FUNCTION_BLOCK Recipe_10010_transportreserve_1
VAR_INPUT
	execute	: BOOL;
	Order	: DUT_RECIPEORDER;
END_VAR
VAR_OUTPUT
	RecipeInfo	: DUT_RECIPEOFFER;
	RecipeDone	: BOOL;	
	InitDone	: BOOL;
END_VAR
VAR
	StepDone	: BOOL;
END_VAR

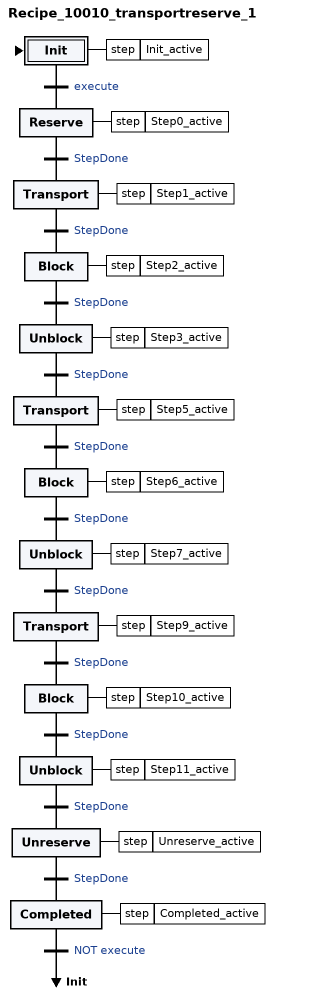
INITIAL_STEP Init:
    Init_active(N);  // step action
END_STEP
TRANSITION FROM Init TO Reserve
    := execute;
END_TRANSITION
STEP Reserve:
    Step0_active(N);  // step action
END_STEP
TRANSITION FROM Reserve TO Transport
    := StepDone;
END_TRANSITION
STEP Transport:
    Step1_active(N);  // step action
END_STEP
TRANSITION FROM Transport TO Block
    := StepDone;
END_TRANSITION
STEP Block:
    Step2_active(N);  // step action
END_STEP
TRANSITION FROM Block TO Unblock
    := StepDone;
END_TRANSITION
STEP Unblock:
    Step3_active(N);  // step action
END_STEP
TRANSITION FROM Unblock TO Transport
    := StepDone;
END_TRANSITION
STEP Transport:
    Step5_active(N);  // step action
END_STEP
TRANSITION FROM Transport TO Block
    := StepDone;
END_TRANSITION
STEP Block:
    Step6_active(N);  // step action
END_STEP
TRANSITION FROM Block TO Unblock
    := StepDone;
END_TRANSITION
STEP Unblock:
    Step7_active(N);  // step action
END_STEP
TRANSITION FROM Unblock TO Transport
    := StepDone;
END_TRANSITION
STEP Transport:
    Step9_active(N);  // step action
END_STEP
TRANSITION FROM Transport TO Block
    := StepDone;
END_TRANSITION
STEP Block:
    Step10_active(N);  // step action
END_STEP
TRANSITION FROM Block TO Unblock
    := StepDone;
END_TRANSITION
STEP Unblock:
    Step11_active(N);  // step action
END_STEP
TRANSITION FROM Unblock TO Unreserve
    := StepDone;
END_TRANSITION
STEP Unreserve:
    Unreserve_active(N);  // step action
END_STEP
TRANSITION FROM Unreserve TO Completed
    := StepDone;
END_TRANSITION
STEP Completed:
    Completed_active(N);  // step action
END_STEP
TRANSITION FROM Completed TO Init
    := NOT execute;
END_TRANSITION

ACTION Block_active:
StepDone := FALSE;

//Skill auswählen
ExecuteSkill.SkillID 		:= 1315;
ExecuteSkill.SkillName	 	:= 'Block';

//Parameter setzen

ExecuteSkill.Parameter[1].ID := 1;
ExecuteSkill.Parameter[1].Name := 'TaskID';
ExecuteSkill.Parameter[1].Value := 124;


(*
ExecuteSkill.Parameter[2].ID := ;
ExecuteSkill.Parameter[2].Name := '';
ExecuteSkill.Parameter[2].Value := ;
*)

(*
ExecuteSkill.Parameter[3].ID := ;
ExecuteSkill.Parameter[3].Name := '';
ExecuteSkill.Parameter[3].Value := ;
*)

(*
ExecuteSkill.Parameter[4].ID := ;
ExecuteSkill.Parameter[4].Name := '';
ExecuteSkill.Parameter[4].Value := ;
*)

(*
ExecuteSkill.Parameter[5].ID := ;
ExecuteSkill.Parameter[5].Name := '';
ExecuteSkill.Parameter[5].Value := ;
*)



ExecuteSkill();

StepDone := ExecuteSkill.Done;
END_ACTION

ACTION Unreserve_active:
StepDone := FALSE;

//Skill auswählen
ExecuteSkill.SkillID 		:= 1311;
ExecuteSkill.SkillName	 	:= 'Unreserve';

//Parameter setzen

ExecuteSkill.Parameter[1].ID := 1;
ExecuteSkill.Parameter[1].Name := 'TaskID';
ExecuteSkill.Parameter[1].Value := 131;


(*
ExecuteSkill.Parameter[2].ID := ;
ExecuteSkill.Parameter[2].Name := '';
ExecuteSkill.Parameter[2].Value := ;
*)

(*
ExecuteSkill.Parameter[3].ID := ;
ExecuteSkill.Parameter[3].Name := '';
ExecuteSkill.Parameter[3].Value := ;
*)

(*
ExecuteSkill.Parameter[4].ID := ;
ExecuteSkill.Parameter[4].Name := '';
ExecuteSkill.Parameter[4].Value := ;
*)

(*
ExecuteSkill.Parameter[5].ID := ;
ExecuteSkill.Parameter[5].Name := '';
ExecuteSkill.Parameter[5].Value := ;
*)



ExecuteSkill();

StepDone := ExecuteSkill.Done;
END_ACTION

ACTION Unblock_active:
StepDone := FALSE;

//Skill auswählen
ExecuteSkill.SkillID 		:= 1316;
ExecuteSkill.SkillName	 	:= 'Unblock';

//Parameter setzen

ExecuteSkill.Parameter[1].ID := 1;
ExecuteSkill.Parameter[1].Name := 'TaskID';
ExecuteSkill.Parameter[1].Value := 125;


(*
ExecuteSkill.Parameter[2].ID := ;
ExecuteSkill.Parameter[2].Name := '';
ExecuteSkill.Parameter[2].Value := ;
*)

(*
ExecuteSkill.Parameter[3].ID := ;
ExecuteSkill.Parameter[3].Name := '';
ExecuteSkill.Parameter[3].Value := ;
*)

(*
ExecuteSkill.Parameter[4].ID := ;
ExecuteSkill.Parameter[4].Name := '';
ExecuteSkill.Parameter[4].Value := ;
*)

(*
ExecuteSkill.Parameter[5].ID := ;
ExecuteSkill.Parameter[5].Name := '';
ExecuteSkill.Parameter[5].Value := ;
*)



ExecuteSkill();

StepDone := ExecuteSkill.Done;
END_ACTION

ACTION Transport1_active:
StepDone := FALSE;

//Skill auswählen
ExecuteSkill.SkillID 		:= 1320;
ExecuteSkill.SkillName	 	:= 'Name';

//Parameter setzen

ExecuteSkill.Parameter[1].ID := 3;
ExecuteSkill.Parameter[1].Name := 'Velocity';
ExecuteSkill.Parameter[1].Value := 2500;



ExecuteSkill.Parameter[2].ID := 4 ;
ExecuteSkill.Parameter[2].Name := 'Acceleration';
ExecuteSkill.Parameter[2].Value := 1000 ;



ExecuteSkill.Parameter[3].ID := 1;
ExecuteSkill.Parameter[3].Name := 'TargetPosition X';
ExecuteSkill.Parameter[3].Value := 3200 ;



ExecuteSkill.Parameter[4].ID := 2;
ExecuteSkill.Parameter[4].Name := 'TargetPosition Z';
ExecuteSkill.Parameter[4].Value := 65 ;


(*
ExecuteSkill.Parameter[5].ID := ;
ExecuteSkill.Parameter[5].Name := '';
ExecuteSkill.Parameter[5].Value := ;
*)



ExecuteSkill();

StepDone := ExecuteSkill.Done;
END_ACTION

ACTION Block1_active:
StepDone := FALSE;

//Skill auswählen
ExecuteSkill.SkillID 		:= 1315;
ExecuteSkill.SkillName	 	:= 'Block';

//Parameter setzen

ExecuteSkill.Parameter[1].ID := 1;
ExecuteSkill.Parameter[1].Name := 'TaskID';
ExecuteSkill.Parameter[1].Value := 127;


(*
ExecuteSkill.Parameter[2].ID := ;
ExecuteSkill.Parameter[2].Name := '';
ExecuteSkill.Parameter[2].Value := ;
*)

(*
ExecuteSkill.Parameter[3].ID := ;
ExecuteSkill.Parameter[3].Name := '';
ExecuteSkill.Parameter[3].Value := ;
*)

(*
ExecuteSkill.Parameter[4].ID := ;
ExecuteSkill.Parameter[4].Name := '';
ExecuteSkill.Parameter[4].Value := ;
*)

(*
ExecuteSkill.Parameter[5].ID := ;
ExecuteSkill.Parameter[5].Name := '';
ExecuteSkill.Parameter[5].Value := ;
*)



ExecuteSkill();

StepDone := ExecuteSkill.Done;
END_ACTION

ACTION Reserve_active:
StepDone := FALSE;
RecipeDone := FALSE;
//Skill auswählen
ExecuteSkill.SkillID 		:= 1310;
ExecuteSkill.SkillName	 	:= 'Reserve';

//Parameter setzen

ExecuteSkill.Parameter[1].ID := 1;
ExecuteSkill.Parameter[1].Name := 'TaskID';
ExecuteSkill.Parameter[1].Value := 123;


(*
ExecuteSkill.Parameter[2].ID := ;
ExecuteSkill.Parameter[2].Name := '';
ExecuteSkill.Parameter[2].Value := ;
*)

(*
ExecuteSkill.Parameter[3].ID := ;
ExecuteSkill.Parameter[3].Name := '';
ExecuteSkill.Parameter[3].Value := ;
*)

(*
ExecuteSkill.Parameter[4].ID := ;
ExecuteSkill.Parameter[4].Name := '';
ExecuteSkill.Parameter[4].Value := ;
*)

(*
ExecuteSkill.Parameter[5].ID := ;
ExecuteSkill.Parameter[5].Name := '';
ExecuteSkill.Parameter[5].Value := ;
*)



ExecuteSkill();

StepDone := ExecuteSkill.Done;
END_ACTION

ACTION Completed_active:
RecipeDone := TRUE;
StepDone := FALSE;
END_ACTION

ACTION Unblock1_active:
StepDone := FALSE;

//Skill auswählen
ExecuteSkill.SkillID 		:= 1316;
ExecuteSkill.SkillName	 	:= 'Unblock';

//Parameter setzen

ExecuteSkill.Parameter[1].ID := 1;
ExecuteSkill.Parameter[1].Name := 'TaskID';
ExecuteSkill.Parameter[1].Value := 128 ;


(*
ExecuteSkill.Parameter[2].ID := ;
ExecuteSkill.Parameter[2].Name := '';
ExecuteSkill.Parameter[2].Value := ;
*)

(*
ExecuteSkill.Parameter[3].ID := ;
ExecuteSkill.Parameter[3].Name := '';
ExecuteSkill.Parameter[3].Value := ;
*)

(*
ExecuteSkill.Parameter[4].ID := ;
ExecuteSkill.Parameter[4].Name := '';
ExecuteSkill.Parameter[4].Value := ;
*)

(*
ExecuteSkill.Parameter[5].ID := ;
ExecuteSkill.Parameter[5].Name := '';
ExecuteSkill.Parameter[5].Value := ;
*)



ExecuteSkill();

StepDone := ExecuteSkill.Done;
END_ACTION

ACTION Transport2_active:
StepDone := FALSE;

//Skill auswählen
ExecuteSkill.SkillID 		:= 1320;
ExecuteSkill.SkillName	 	:= 'Transport';

//Parameter setzen

ExecuteSkill.Parameter[1].ID := 3;
ExecuteSkill.Parameter[1].Name := 'Velocity';
ExecuteSkill.Parameter[1].Value := 2800;



ExecuteSkill.Parameter[2].ID :=  1;
ExecuteSkill.Parameter[2].Name := 'TargetPosition X';
ExecuteSkill.Parameter[2].Value := 200 ;



ExecuteSkill.Parameter[3].ID := 2;
ExecuteSkill.Parameter[3].Name := 'TargetPosition Z';
ExecuteSkill.Parameter[3].Value := 35 ;



ExecuteSkill.Parameter[4].ID := 4;
ExecuteSkill.Parameter[4].Name := 'Acceleration';
ExecuteSkill.Parameter[4].Value := 2000 ;


(*
ExecuteSkill.Parameter[5].ID := ;
ExecuteSkill.Parameter[5].Name := '';
ExecuteSkill.Parameter[5].Value := ;
*)



ExecuteSkill();

StepDone := ExecuteSkill.Done;
END_ACTION

ACTION Block2_active:
StepDone := FALSE;

//Skill auswählen
ExecuteSkill.SkillID 		:= 1315;
ExecuteSkill.SkillName	 	:= 'Block';

//Parameter setzen

ExecuteSkill.Parameter[1].ID := 1;
ExecuteSkill.Parameter[1].Name := 'TaskID';
ExecuteSkill.Parameter[1].Value := 130;


(*
ExecuteSkill.Parameter[2].ID := ;
ExecuteSkill.Parameter[2].Name := '';
ExecuteSkill.Parameter[2].Value := ;
*)

(*
ExecuteSkill.Parameter[3].ID := ;
ExecuteSkill.Parameter[3].Name := '';
ExecuteSkill.Parameter[3].Value := ;
*)

(*
ExecuteSkill.Parameter[4].ID := ;
ExecuteSkill.Parameter[4].Name := '';
ExecuteSkill.Parameter[4].Value := ;
*)

(*
ExecuteSkill.Parameter[5].ID := ;
ExecuteSkill.Parameter[5].Name := '';
ExecuteSkill.Parameter[5].Value := ;
*)



ExecuteSkill();

StepDone := ExecuteSkill.Done;
END_ACTION

ACTION Transport_active:
StepDone := FALSE;

//Skill auswählen
ExecuteSkill.SkillID 		:= 1320;
ExecuteSkill.SkillName	 	:= 'Transport';

//Parameter setzen

ExecuteSkill.Parameter[1].ID :=3 ;
ExecuteSkill.Parameter[1].Name := 'Velocity';
ExecuteSkill.Parameter[1].Value := 3000;



ExecuteSkill.Parameter[2].ID :=1 ;
ExecuteSkill.Parameter[2].Name := 'TargetPosition X';
ExecuteSkill.Parameter[2].Value := 2000;



ExecuteSkill.Parameter[3].ID := 2 ;
ExecuteSkill.Parameter[3].Name := 'TargetPosition Z';
ExecuteSkill.Parameter[3].Value := 55 ;



ExecuteSkill.Parameter[4].ID := 4 ;
ExecuteSkill.Parameter[4].Name := 'Acceleration';
ExecuteSkill.Parameter[4].Value := 1500;


(*
ExecuteSkill.Parameter[5].ID := ;
ExecuteSkill.Parameter[5].Name := '';
ExecuteSkill.Parameter[5].Value := ;
*)



ExecuteSkill();

StepDone := ExecuteSkill.Done;
END_ACTION

ACTION Init_active:
RecipeDone := FALSE;

// Initialisation of Recipe Parameters an name etc
RecipeInfo.Name := 'Sample Product Name';
RecipeInfo.Description := 'This Recipe produces a product, which is very productive';
RecipeInfo.Dummy := FALSE;
RecipeInfo.RecipeID := 10000; 	// 
Initdone := TRUE;

//Parameter 1:
(*
	RecipeInfo.UserParameter[1].Dummy 		:= 
	RecipeInfo.UserParameter[1].Default		:=
	RecipeInfo.UserParameter[1].Description	:=
	RecipeInfo.UserParameter[1].MaxValue	:=
	RecipeInfo.UserParameter[1].MinValue	:=
	RecipeInfo.UserParameter[1].Name		:=
	RecipeInfo.UserParameter[1].Unit		:=
*)
//Parameter 2:

(*
	RecipeInfo.UserParameter[2].Dummy 		:= 
	RecipeInfo.UserParameter[2].Default		:=
	RecipeInfo.UserParameter[2].Description	:=
	RecipeInfo.UserParameter[2].MaxValue	:=
	RecipeInfo.UserParameter[2].MinValue	:=
	RecipeInfo.UserParameter[2].Name		:=
	RecipeInfo.UserParameter[2].Unit		:=
*)

//Parameter 3:

(*
	RecipeInfo.UserParameter[3].Dummy 		:= 
	RecipeInfo.UserParameter[3].Default		:=
	RecipeInfo.UserParameter[3].Description	:=
	RecipeInfo.UserParameter[3].MaxValue	:=
	RecipeInfo.UserParameter[3].MinValue	:=
	RecipeInfo.UserParameter[3].Name		:=
	RecipeInfo.UserParameter[3].Unit		:=
*)

//Parameter 4:

(*
	RecipeInfo.UserParameter[4].Dummy 		:= 
	RecipeInfo.UserParameter[4].Default		:=
	RecipeInfo.UserParameter[4].Description	:=
	RecipeInfo.UserParameter[4].MaxValue	:=
	RecipeInfo.UserParameter[4].MinValue	:=
	RecipeInfo.UserParameter[4].Name		:=
	RecipeInfo.UserParameter[4].Unit		:=
*)


//Parameter 5:

(*
	RecipeInfo.UserParameter[5].Dummy 		:= 
	RecipeInfo.UserParameter[5].Default		:=
	RecipeInfo.UserParameter[5].Description	:=
	RecipeInfo.UserParameter[5].MaxValue	:=
	RecipeInfo.UserParameter[5].MinValue	:=
	RecipeInfo.UserParameter[5].Name		:=
	RecipeInfo.UserParameter[5].Unit		:=
*)
END_ACTION

ACTION Unblock2_active:
StepDone := FALSE;

//Skill auswählen
ExecuteSkill.SkillID 		:= 1316;
ExecuteSkill.SkillName	 	:= 'Unblock';

//Parameter setzen

ExecuteSkill.Parameter[1].ID := 1;
ExecuteSkill.Parameter[1].Name := 'TaskID';
ExecuteSkill.Parameter[1].Value := 131;


(*
ExecuteSkill.Parameter[2].ID := ;
ExecuteSkill.Parameter[2].Name := '';
ExecuteSkill.Parameter[2].Value := ;
*)

(*
ExecuteSkill.Parameter[3].ID := ;
ExecuteSkill.Parameter[3].Name := '';
ExecuteSkill.Parameter[3].Value := ;
*)

(*
ExecuteSkill.Parameter[4].ID := ;
ExecuteSkill.Parameter[4].Name := '';
ExecuteSkill.Parameter[4].Value := ;
*)

(*
ExecuteSkill.Parameter[5].ID := ;
ExecuteSkill.Parameter[5].Name := '';
ExecuteSkill.Parameter[5].Value := ;
*)



ExecuteSkill();

StepDone := ExecuteSkill.Done;
END_ACTION

END_FUNCTION_BLOCK

(* stored: Version 1.1.0.1, ProductVersion 3.1.0.25
   POU Recipe_10010_transportreserve_1: Id {49c20850-82e6-41db-af83-78d750b4b527}
   Action Block_active: Id {0622d7c7-c24b-4408-99b4-3c3ab982b649}
   Action Unreserve_active: Id {132797b3-3f11-4448-805c-06e64fec2dbf}
   Action Unblock_active: Id {1608981b-0d1b-472d-a4da-fb8fe1cba0b8}
   Action Transport1_active: Id {5251e6ef-3639-45f4-a658-d869b584a69a}
   Action Block1_active: Id {58286793-674e-49d6-bbfc-cd378cd91a7f}
   Action Reserve_active: Id {67a7a822-2df2-46b3-803c-7ae15455056d}
   Action Completed_active: Id {8866b812-0e9a-4a7d-9b35-57f7ef80a4fe}
   Action Unblock1_active: Id {9109b334-ffc6-498f-bc10-004839868031}
   Action Transport2_active: Id {9c74856b-8ad3-4214-97db-5be9f009f81b}
   Action Block2_active: Id {acae7adc-11a8-45a2-9d65-7b3818b91fca}
   Action Transport_active: Id {d374ce22-e328-4ce2-aff9-67aa4d69e719}
   Action Init_active: Id {d3b94830-34a1-41cf-9d05-10ab9e573a35}
   Action Unblock2_active: Id {f11bcb05-259a-40b1-9b1c-1a387d32ac9b} *)
